{attribute 'qualified_only'}
{attribute 'strict'}
TYPE E_ScopeCommand : 
(
	eDefault := 0,
	ePause,
	eStop
) ;
END_TYPE

(* stored: DUT E_ScopeCommand: Id 2bc43781-cfbe-4064-b9d4-01b43e510a9b *)
